// TIA Portal project "oil pump" (V17)
// Problem Statement
// An oil pump should start up after pressing start push button and the main motor will start automatically after 15 sec after pressing stop push button main motor will stop immediately and the oil pump will stop automatically after 15 sec.

(* hardware
DEVICE "S7-1200 station_1"  S7-1200 Station
   slot 0: "Rack_0"  S7-1200 Rack  Rack  V1.0
   slot 1: "PLC_1"  CPU 1212C AC/DC/Rly  6ES7 212-1BE40-0XB0  V4.5
*)

// ===== PLC "PLC_1"  CPU 1212C AC/DC/Rly =====

VAR_GLOBAL   // PLC tag table "Default tag table"
   "PB" AT %I0.0 : Bool;
   "S_PB" AT %I0.1 : Bool;
   "Oil Pump" AT %Q0.0 : Bool;
   "Main motor" AT %Q0.1 : Bool;
   "Tag_1" AT %MD0 : Time;
   "Tag_2" AT %MD1 : Time;
END_VAR

// folder: System blocks/Program resources

DATA_BLOCK "IEC_Timer_0_DB_1"   // DB2
{ S7_Optimized_Access := 'TRUE' }
AUTHOR : Simatic
FAMILY : IEC
NAME : IEC_TMR
VERSION : 1.0
// stored: InstanceOfName IEC_TIMER
"IEC_TIMER"
BEGIN
END_DATA_BLOCK

DATA_BLOCK "IEC_Timer_0_DB_2"   // DB3
{ S7_Optimized_Access := 'TRUE' }
AUTHOR : Simatic
FAMILY : IEC
NAME : IEC_TMR
VERSION : 1.0
// stored: InstanceOfName IEC_TIMER
"IEC_TIMER"
BEGIN
END_DATA_BLOCK

// folder: (top level)

ORGANIZATION_BLOCK "Main"   // OB1, LAD, ProgramCycle
TITLE = "Main Program Sweep (Cycle)"
{ S7_Optimized_Access := 'TRUE' }
VERSION : 0.1
   VAR_INPUT
      Initial_Call : Bool;   // Initial call of this OB
      Remanence : Bool;   // =True, if remanent data are available
   END_VAR
   VAR_TEMP   // added for the SCL form of the ladder/FBD networks
      _w1 : Bool;
   END_VAR
BEGIN

REGION Network 1
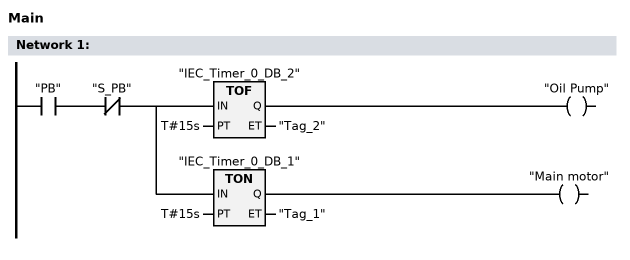
   #_w1 := "PB" AND NOT "S_PB";
   "IEC_Timer_0_DB_2".TOF(IN := #_w1, PT := T#15s, ET => "Tag_2");
   "Oil Pump" := "IEC_Timer_0_DB_2".Q;
   "IEC_Timer_0_DB_1".TON(IN := #_w1, PT := T#15s, ET => "Tag_1");
   "Main motor" := "IEC_Timer_0_DB_1".Q;
END_REGION
END_ORGANIZATION_BLOCK